FUNCTION_BLOCK IndexMoverSequence EXTENDS CyclicBase
VAR
	State : IndexSequenceState;  
	CurrentStation : UINT;
	TargetStationPosition : MC_LREAL;
	_MoverVelocity : MC_LREAL := 1000.0;
	stSequenceInfo : MoverSequenceInfo;
	StationArray : ARRAY[1..SystemParameters.NumberOfStations] OF IProcess;
	ThisMover : I_XtsMoverAxis;
	StateMachine : IPmlStateMachine;
	_startPosition : MC_LREAL;
	_XtsNoHome : BOOL;
	_NonModuloMoves : BOOL := false;
END_VAR

{analysis -2}

METHOD Abort : BOOL
VAR_INPUT
END_VAR
State := IndexSequenceState.Available;
CurrentStation := 0;
TargetStationPosition := 0.0;
stSequenceInfo.CurrentStation := UINT_TO_INT(CurrentStation);
stSequenceInfo.MoverId := ThisMover.AxisRef.NcToPlc.AxisId;
stSequenceInfo.State := State;
stSequenceInfo.Velocity := ThisMover.AxisRef.NcToPlc.ActVelo;
Abort := TRUE;
END_METHOD

METHOD PUBLIC  Cycle : HRESULT
VAR_INPUT
END_VAR
IF StateMachine.GetCurrentState() = E_PMLState.ePMLState_Aborting THEN
	State := IndexSequenceState.Aborting;
ELSIF StateMachine.GetCurrentState() = E_PMLState.ePMLState_Stopping THEN
	State := IndexSequenceState.Stopping;
END_IF
Cycle := S_OK;
CASE State OF
	IndexSequenceState.Init:
		IF ThisMover.isMoverDetected() THEN
			State := IndexSequenceState.Available;
		END_IF
		
	IndexSequenceState.Available:
		IF StateMachine.GetCurrentState() = E_PMLState.ePMLState_Execute THEN
			State := IndexSequenceState.MovingToStart;
		END_IF
		
	IndexSequenceState.MovingToStart:
		IF ThisMover.isMoverAtPosition(position := _startPosition) OR _XtsNoHome THEN
			State := IndexSequenceState.AtStart;
		END_IF
			
	IndexSequenceState.AtStart:
		IF StationArray[1].IsReady() THEN
			State := IndexSequenceState.GetNextMove;
		END_IF

	IndexSequenceState.MovingToStation:
		IF ThisMover.isMoverStationary() THEN 
			IF ThisMover.isMoverAtPosition(TargetStationPosition) THEN
				IF StationArray[CurrentStation].IsProcess THEN
					State := IndexSequenceState.AtProcess;
				ELSE
					State := IndexSequenceState.AtStation;
				END_IF
				StationArray[CurrentStation].HasMover(ThisMover);
			ELSE
				State := IndexSequenceState.QueuedAtStation;
			END_IF
		END_IF
		
	IndexSequenceState.QueuedAtStation:
		IF NOT ThisMover.isMoverStationary() THEN
				State := IndexSequenceState.MovingToStation;
		END_IF

	IndexSequenceState.AtStation:
		IF StationArray[CurrentStation].isComplete() THEN
			State := IndexSequenceState.GetNextMove;
		END_IF

	IndexSequenceState.AtProcess:
		ThisMover.MoveTo(RequiredPosition := StationArray[CurrentStation].EndPosition,
								MoveVelocity := StationArray[CurrentStation].ProcessVelocity,
								NonModuloMove := _NonModuloMoves);
		State := IndexSequenceState.InProcess;
								
	IndexSequenceState.InProcess:
		IF ThisMover.isMoverStationary() THEN 
			IF ThisMover.isMoverAtPosition(StationArray[CurrentStation].EndPosition) THEN
				State := IndexSequenceState.GetNextMove;
			END_IF
		END_IF
	
	IndexSequenceState.GetNextMove:
		IF CurrentStation = SystemParameters.NumberOfStations THEN
			IF ThisMover.MoveTo(RequiredPosition := _startPosition,
							MoveVelocity := _MoverVelocity,
							NonModuloMove := _NonModuloMoves) = 1 THEN
				State := IndexSequenceState.MovingToStart;
				StationArray[CurrentStation].MoverAway();
				CurrentStation := 0; 
			END_IF
		ELSE
			State := IndexSequenceState.GoToNextStation;
		END_IF
		
	IndexSequenceState.GoToNextStation:
		IF StationArray[CurrentStation + 1].IsProcess THEN
			TargetStationPosition := StationArray[CurrentStation + 1].StartPosition;
		ELSE
			TargetStationPosition := StationArray[CurrentStation + 1].Position;
		END_IF
		IF 	ThisMover.MoveTo(RequiredPosition := TargetStationPosition,
							MoveVelocity := _MoverVelocity,
							NonModuloMove := _NonModuloMoves) = 1 THEN
			IF CurrentStation <> 0 THEN
				StationArray[CurrentStation].MoverAway();	
			END_IF		
			CurrentStation := CurrentStation + 1;
			State := IndexSequenceState.MovingToStation;
		END_IF	

	IndexSequenceState.Stopping:
		IF StateMachine.GetCurrentState() = E_PMLState.ePMLState_Stopped THEN
			State := IndexSequenceState.Available;
			CurrentStation := 0;
			TargetStationPosition := 0.0;
		END_IF			
		
	IndexSequenceState.Aborting:
		IF StateMachine.GetCurrentState() = E_PMLState.ePMLState_Aborted THEN
			State := IndexSequenceState.Available;
			CurrentStation := 0;
			TargetStationPosition := 0.0;
		END_IF
	ELSE
		Cycle := E_FAIL;
END_CASE

//Cyclic update info data
stSequenceInfo.CurrentStation := UINT_TO_INT(CurrentStation);
stSequenceInfo.MoverId := ThisMover.AxisRef.NcToPlc.AxisId;
stSequenceInfo.State := State;
stSequenceInfo.Velocity := ThisMover.AxisRef.NcToPlc.ActVelo;
END_METHOD

METHOD FB_init : BOOL
VAR_INPUT
	bInitRetains : BOOL; // if TRUE, the retain variables are initialized (warm start / cold start)
	bInCopyCode : BOOL;  // if TRUE, the instance afterwards gets moved into the copy code (online change)
	XtsRunner : I_ObjectRunner;
END_VAR
XtsRunner.RegisterModule(THIS^);
END_METHOD

PROPERTY MoverVelocity : mc_lreal
GET
MoverVelocity := _MoverVelocity;
END_GET
SET
_MoverVelocity := MoverVelocity;
END_SET
END_PROPERTY

PROPERTY MyMover : I_XtsMoverAxis
GET
MyMover := ThisMover;
END_GET
SET
ThisMover := MyMover;
END_SET
END_PROPERTY

PROPERTY MyStartPosition : MC_LREAL
GET
MyStartPosition := _startPosition;
END_GET
SET
_startPosition := MyStartPosition;
END_SET
END_PROPERTY

PROPERTY MyStateMachine : IPmlStateMachine
GET
MyStateMachine := StateMachine;
END_GET
SET
StateMachine := MyStateMachine;
END_SET
END_PROPERTY

PROPERTY MyStations : ARRAY[1..SystemParameters.NumberOfStations] OF IProcess
GET
MyStations := StationArray;
END_GET
SET
StationArray := MyStations;
END_SET
END_PROPERTY

PROPERTY XtsNoHome : BOOL
GET
XtsNoHome := _XtsNoHome;
END_GET
SET
_XtsNoHome := XtsNoHome;
END_SET
END_PROPERTY

END_FUNCTION_BLOCK

(* stored: Version 1.1.0.1, ProductVersion 3.1.4026.11
   POU IndexMoverSequence: Id {50af290e-a0d7-45b3-a647-c8828b096bd1}, SpecialFunc None
   Method Abort: Id {01dd3306-e903-4754-85c4-ea13c41e0b8c}
   Method Cycle: Id {0bc270b2-0e7a-4545-b872-87f2d15ca3f5}
   Method FB_init: Id {b89bce77-cfe9-4671-96f6-b6944812f4ae}
   Property MoverVelocity: Id {4f2224ad-0534-4bd9-a8e4-5b63b7e53b5c}
   Get Get: Id {0bf3cfa6-cc44-4232-989f-70bced017a55}
   Set Set: Id {a9bdfb5a-ef56-4b9e-9f78-288684e24d6c}
   Property MyMover: Id {d0dbd650-93c6-4e7f-a733-abc40a2f12bf}
   Get Get: Id {52e46adf-1b9f-404f-a8d7-de686d91d4ef}
   Set Set: Id {a9693a81-065c-4ba2-8a99-3606c71cf06a}
   Property MyStartPosition: Id {30ed087d-d896-49f8-aaff-c511c0d55a71}
   Get Get: Id {ebcb0d89-302c-4f5d-86e5-f5e15f136ea5}
   Set Set: Id {57b76837-f6ca-44d6-8033-7a2d9ee3e944}
   Property MyStateMachine: Id {d844989e-66dd-4349-8c85-edbcb74c9dc3}
   Get Get: Id {2d0a1e27-5c9e-4b26-a4e6-24217a260482}
   Set Set: Id {a96c0464-f76e-4411-81f3-99766fd72773}
   Property MyStations: Id {d7be010f-02ed-44eb-9206-f5e1204f6ead}
   Get Get: Id {b9858861-0750-4c3d-b2e9-7dc3a973373a}
   Set Set: Id {7371b464-f457-4be2-b93c-2c3bb66d5175}
   Property XtsNoHome: Id {7aad9af3-71dc-4b8d-9a2b-19016c2a644b}
   Get Get: Id {d3413585-01ef-4909-a612-e4cda3a7b8e0}
   Set Set: Id {ca6f67d3-9265-4c0f-849c-5e4c98f82e9b} *)
